FUNCTION_BLOCK MKS_275_to_500_HvOn
VAR_INPUT
	stPirani	:	ST_MKS_275;
END_VAR
VAR_OUTPUT
END_VAR
VAR_IN_OUT
	stCC		:	ST_MKS_500;
END_VAR
VAR
END_VAR

(* HV ON for MKS 275 Pirani Gauge to Turn on MKS 500 Cold Cathode Gauge
A. Pai 
2/8/2017


Takes in Pirani Gauge as an INPUT and Cold Cathode gauge as an IN_OUT. 
The Cold Cathode uses the Pirani Pressure to determine whether or not
to turn on or turn off. 

There is no turn on/ turn off timer. 
No Hysterisis either. 

Turn on timer is left to Cold Cathode Function Block.
*)
//The Cold Cathode Setpoint is 0.01 Torr
IF stPirani.rPress <= 1.0E-2 THEN
	stCC.i_xHvOn := TRUE;//Turn on Cathode
ELSE
	stCC.i_xHvOn := FALSE;//Turn off Cathode
END_IF

END_FUNCTION_BLOCK

(* stored: Version 1.1.0.1, ProductVersion 3.1.4020.12
   POU MKS_275_to_500_HvOn: Id {c90aa29b-b222-4340-83a6-1c3483b75837}, SpecialFunc None *)
